(* IEC 61131-3 sources: RL_MAR/experiments/comparison/llm4plc/results/gpt-4o_20260507_114630/20260507_115734, 1 file *)

(* ---- generated_code_iteration_0.st ---- *)
plaintext
START_ST
FUNCTION_BLOCK FlowerArrangingMachine
VAR_INPUT
    FlowerTypeSensor : INT; (* Input for detecting flower type *)
    FlowerColorSensor : INT; (* Input for detecting flower color *)
END_VAR
VAR_OUTPUT
    ArrangingMechanism : INT; (* Output for controlling arranging mechanism *)
    ConveyorBelt : BOOL; (* Output for controlling conveyor belt *)
END_VAR
VAR
    state : INT; (* Internal state variable *)
    prevState : INT; (* Internal variable to track the previous state *)
END_VAR

(* Logic for state transitions and outputs *)
IF FlowerTypeSensor = 1 AND FlowerColorSensor = 1 THEN
    state := 1; (* Processing type 1 red flower *)
ELSIF FlowerTypeSensor = 1 AND FlowerColorSensor = 2 THEN
    state := 2; (* Processing type 1 blue flower *)
ELSIF FlowerTypeSensor = 2 AND FlowerColorSensor = 1 THEN
    state := 3; (* Processing type 2 red flower *)
ELSIF FlowerTypeSensor = 2 AND FlowerColorSensor = 2 THEN
    state := 4; (* Processing type 2 blue flower *)
ELSE
    state := 5; (* Invalid flower type or color *)
END_IF

(* State handling and output logic *)
CASE state OF
    0: (* IDLE state *)
        ArrangingMechanism := 0;
        ConveyorBelt := FALSE;
    1: (* Processing type 1 red flower *)
        ArrangingMechanism := 1;
        ConveyorBelt := TRUE;
    2: (* Processing type 1 blue flower *)
        ArrangingMechanism := 2;
        ConveyorBelt := TRUE;
    3: (* Processing type 2 red flower *)
        ArrangingMechanism := 3;
        ConveyorBelt := TRUE;
    4: (* Processing type 2 blue flower *)
        ArrangingMechanism := 4;
        ConveyorBelt := TRUE;
    5: (* Invalid flower type or color *)
        ArrangingMechanism := 0;
        ConveyorBelt := FALSE;
END_CASE

(* Reset state to IDLE at the end of the cycle *)
prevState := state;
state := 0;

END_FUNCTION_BLOCK
END_ST
